Staubli VAL3: loadmaster0.pgx

program loadmaster0(string x_sMasterFile0)
begin
  if master:libLoad(x_sMasterFile0)<0
    popUpMsg("nO ok")
  endIf
  //由于mastercam生成出来的真实坐标位置是保存在tTool里的。
  frmaster[0].trsf=master:tTool.trsf
  //取个数
  nsize[0]=size(master:ptRoutingPath)
  //存个数
  resize(pdemo0,1,nsize[0])
  //保存程序
  master:libSave()
end
